INTERFACE ITF_Actuator_HMI_Init EXTENDS ITF_BaseControlElement, ITF_Actuator_HMI_Connector

END_INTERFACE

(* stored: Version 1.1.0.1
   Itf ITF_Actuator_HMI_Init: Id {be35956d-b830-40ec-8943-cdb892bafda0} *)
